FUNCTION_BLOCK FB_LensSet EXTENDS FB_Fallible IMPLEMENTS I_LensSet
VAR
    fbRadius : FB_QuantityLREALPublic(Units := 'm');
    fbLens : FB_Lens;

    afbLens : ARRAY [1..GVL_Physics.nMaxNumLensesInSet] OF FB_Lens;
    nNumLenses : INT;
END_VAR


METHOD GetLens
VAR_INPUT
    LensNum	: INT;
END_VAR
VAR_IN_OUT
    Lens	: FB_Lens;
END_VAR

ClearError();

IF NOT IndexInRange(LensNum) THEN
    SetError(Msg := IndexOutOfRangeErrorMsg(nLensNum := LensNum));
    RETURN;
END_IF

Lens := afbLens[LensNum];
END_METHOD


METHOD IndexInRange : BOOL
VAR_INPUT
    nIndex : INT;
END_VAR

IndexInRange := nIndex > 0 AND nIndex <= NumLenses;
END_METHOD


METHOD IndexOutOfRangeErrorMsg : T_MaxString
VAR_INPUT
    nLensNum : INT;
END_VAR

IndexOutOfRangeErrorMsg :=
        CONCAT('Requested index is out of the allowable range. ',
        CONCAT('0 < [',
        CONCAT(INT_TO_STRING(nLensNum),
        CONCAT('] <= ',
        CONCAT(INT_TO_STRING(NumLenses),
        ' is not true.')))));
END_METHOD


PROPERTY NumLenses : INT
GET

NumLenses := nNumLenses;
END_GET
SET

IF NumLenses > 0 AND NumLenses <= GVL_Physics.nMaxNumLensesInSet THEN
    nNumLenses := NumLenses;
ELSE
    SetError(Msg := CONCAT('Attempted to set number of lenses to: [',
        CONCAT(INT_TO_STRING(NumLenses),
        CONCAT('] which does not meet the criteria: 0 < NumLenses <= GVL_Physics.nMaxNumLensesInSet = [',
        CONCAT(INT_TO_STRING(GVL_Physics.nMaxNumLensesInSet),
        ']'))))
    );
END_IF
END_SET
END_PROPERTY


METHOD SetLens
VAR_INPUT
    Lens : I_Lens;
    LensNum : INT;
END_VAR

ClearError();

IF NOT IndexInRange(LensNum) THEN
    SetError(Msg := IndexOutOfRangeErrorMsg(nLensNum := LensNum));
    RETURN;
END_IF

fbLens.Copy(Lens);

IF fbLens.GetError() THEN
    SetError(
        Msg := CONCAT('The input lens has the following error message: [',
        CONCAT(fbLens.GetErrorMsg(),
        ']'))
    );
    RETURN;
END_IF

afbLens[LensNum] := fbLens;
END_METHOD

END_FUNCTION_BLOCK

(* stored: Version 1.1.0.1
   POU FB_LensSet: Id {9055d704-4d25-40c5-873f-804fc0b293d8}, SpecialFunc None
   Method GetLens: Id {9e1ed0e8-5daa-4afd-85a9-a0c8ba1a6071}
   Method IndexInRange: Id {736b6ca6-387b-4727-80f6-b6d61a70ddd3}
   Method IndexOutOfRangeErrorMsg: Id {b2d5c30b-5f25-4b92-8eb7-0371b1cc775a}
   Property NumLenses: Id {1ababeff-88b4-4598-8f6f-5898604237f0}
   Get Get: Id {a045bb85-1352-478d-b38c-0658422571a9}
   Set Set: Id {79ab4a51-2bc8-4a47-ab7e-f9e6958d9160}
   Method SetLens: Id {d2a31209-d8ac-4b1d-a13e-7d8ca7bdb34d} *)
